{attribute 'pack_mode' := '1'}
TYPE ST_TcpTask :
STRUCT
	TaskName : STRING(24);
	TaskType : INT; (* 0:Once, 1:Regular *)
	TaskData : ARRAY[0..255] OF BYTE;
END_STRUCT
END_TYPE

(* stored: Version 1.1.0.1, ProductVersion 3.1.4024.12
   DUT ST_TcpTask: Id {5312c90a-8780-4e3a-a50c-3a8f5b55bacd} *)
